// TwinCAT 3 PLC project Main
// ProgramVersion: 3.1.4024.0
// libraries:
//   Tc2_Standard, * (Beckhoff Automation GmbH)
//   Tc2_System, * (Beckhoff Automation GmbH)
//   Tc3_Module, * (Beckhoff Automation GmbH)
// project tree:
//   DUTs/ MyReport.TcDUT, ExampleTableRow.TcDUT
//   / PlcTask.TcTTO
//   POUs/ MAIN.TcPOU
// real-time tasks:
//   TASK PlcTask: cycle T#10ms, priority 20, ADS port 350

CONFIGURATION Main
    RESOURCE PLC ON TwinCAT3
        TASK PlcTask(INTERVAL := T#10ms, PRIORITY := 20);
        PROGRAM MAIN WITH PlcTask : MAIN;
    END_RESOURCE
END_CONFIGURATION

// ---- DUTs/MyReport.TcDUT
TYPE MyReport :
STRUCT
	ExampleString : STRING := 'This is a test string';
	ExampleInt : INT := 12345;
	ExampleTable : ARRAY [0..2] OF ExampleTableRow
		:= [(
			Name:='Example row 1',
			Value:=123
		),(
			Name:='Example row 2',
			Value:=456
		),(
			Name:='Example row 3',
			Value:=789
		)];
END_STRUCT
END_TYPE

// ---- DUTs/ExampleTableRow.TcDUT
TYPE ExampleTableRow :
STRUCT
	Name : STRING;
	Value : INT;
END_STRUCT
END_TYPE

// ---- POUs/MAIN.TcPOU
PROGRAM MAIN
VAR
	myReport : MyReport;
END_VAR

END_PROGRAM
